(* CODESYS project Function_Block.project
   Title: Function_Block
   Version: 0.0.0.0
   Author: MustafaZahid

Project tree, tasks and I/O mapping:
  MyController : TM241C24T/U, Schneider Electric, order no. TM241C24T/U, version 4.0.6.18
    application Application
      task MAST (cyclic, interval 20 ms, priority 15, watchdog 100 ms x 1) calls POU
      global variables GVL
      program POU [LD]
      FB's/
        function block Sensor [LD]
        function block Motion [LD]
    DI : Digital Inputs, Schneider Electric, version 4.0.6.18
        input  iwDI_IW0 : WORD  // IW0
        input  ibDI_IB1 : BYTE  // IB1
    DQ : Digital Outputs, Schneider Electric, version 4.0.6.18
        settings: Outputs Usage = 3
        output qwDQ_QW0 : WORD  // QW0
        output qbDQ_QB1 : BYTE  // QB1
    Counters : Counters, Schneider Electric, version 4.0.6.18
    Pulse_Generators : Pulse Generators, Schneider Electric, version 4.0.6.18
        settings: Instance name = 'Axis_1'; B output History = 'old=-1 new=1'; A output History = 'old=-1 new=0'; Temporary Instance name = 'Axis_1'
    Cartridge_1 : Cartridge, Schneider Electric, version 4.0.6.18
    IO_Bus : IO bus - TM3, Schneider Electric, version 4.0.6.18
    COM_Bus : COM bus, Schneider Electric, version 4.0.6.18
    Serial_Line_1 : Serial line, Schneider Electric, version 4.0.6.18
      SoMachine_Network_Manager : SoMachine-Network Manager, Schneider Electric, version 4.0.0.2
    Serial_Line_2 : Serial line, Schneider Electric, version 4.0.6.18
      Modbus_Manager : Modbus Manager, Schneider Electric, version 4.0.0.2
*)

// MyController/Application/GVL
VAR_GLOBAL
END_VAR

// MyController/Application/POU
PROGRAM POU
VAR
	Motor: BOOL;
	Bending: BOOL;
	Motor_En_1: BOOL;
	Motor_En_2: BOOL;
	Motor_En_3: BOOL;
	Bending_En_1: BOOL;
	Bending_En_2: BOOL;
	Bending_En_3: BOOL;
	Detect_1: BOOL;
	Sensor_1: Sensor;
	Detect_2: BOOL;
	Sensor_2: Sensor;
	Detect_3: BOOL;
	Sensor_3: Sensor;
END_VAR

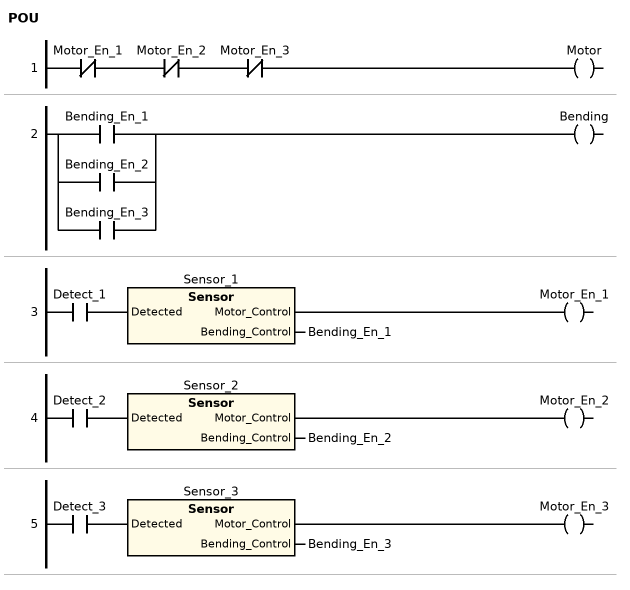
// NETWORK 1
Motor := NOT Motor_En_1 AND NOT Motor_En_2 AND NOT Motor_En_3;

// NETWORK 2
Bending := Bending_En_1 OR Bending_En_2 OR Bending_En_3;

// NETWORK 3
Sensor_1(Detected := Detect_1, Bending_Control => Bending_En_1); // Sensor
Motor_En_1 := Sensor_1.Motor_Control;

// NETWORK 4
Sensor_2(Detected := Detect_2, Bending_Control => Bending_En_2); // Sensor
Motor_En_2 := Sensor_2.Motor_Control;

// NETWORK 5
Sensor_3(Detected := Detect_3, Bending_Control => Bending_En_3); // Sensor
Motor_En_3 := Sensor_3.Motor_Control;

END_PROGRAM

// MyController/Application/FB's/Sensor
FUNCTION_BLOCK Sensor
VAR_INPUT
	Detected: BOOL;
END_VAR
VAR_OUTPUT
	Motor_Control: BOOL;
	Bending_Control: BOOL;
END_VAR
VAR
	TON_0: TON;
	TON_1: TON;
	TON_2: TON;
END_VAR

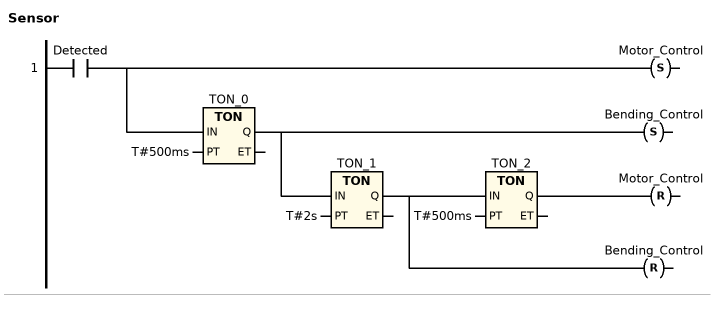
// NETWORK 1
Motor_Control S= Detected;
TON_0(IN := Detected, PT := T#500ms); // TON
Bending_Control S= TON_0.Q;
TON_1(IN := TON_0.Q, PT := T#2s); // TON
TON_2(IN := TON_1.Q, PT := T#500ms); // TON
Motor_Control R= TON_2.Q;
Bending_Control R= TON_1.Q;

END_FUNCTION_BLOCK

// MyController/Application/FB's/Motion
FUNCTION_BLOCK Motion
VAR_INPUT
	Power: BOOL;
END_VAR
VAR_OUTPUT
	Direction_Value: MC_DIRECTION;
END_VAR
VAR
	MC_Power: MC_Power_PTO;
	MC_MoveVelocity: MC_MoveVelocity_PTO;
	Vel_Execute: BOOL;
	Direction: MC_DIRECTION;
	MC_Home: MC_Home_PTO;
	Set_Home: BOOL;
END_VAR

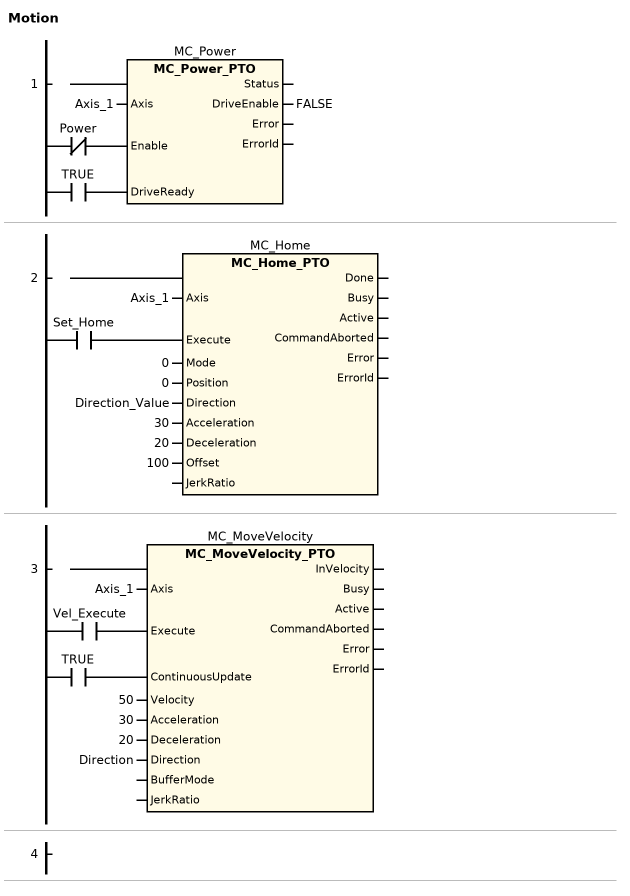
// NETWORK 1
MC_Power(Axis := Axis_1, Enable := NOT Power, DriveReady := TRUE, DriveEnable => FALSE); // MC_Power_PTO

// NETWORK 2
MC_Home(
    Axis := Axis_1,
    Execute := Set_Home,
    Mode := 0,
    Position := 0,
    Direction := Direction_Value,
    Acceleration := 30,
    Deceleration := 20,
    Offset := 100); // MC_Home_PTO

// NETWORK 3
MC_MoveVelocity(
    Axis := Axis_1,
    Execute := Vel_Execute,
    ContinuousUpdate := TRUE,
    Velocity := 50,
    Acceleration := 30,
    Deceleration := 20,
    Direction := Direction); // MC_MoveVelocity_PTO

// NETWORK 4

END_FUNCTION_BLOCK
